(* CODESYS project Flight Simulator_RECOVERED_2024-10-07T14-12-38.project

Project tree, tasks and I/O mapping:
  PLC : HX-CP1S08, Hitachi Industrial Equipment Systems Co., Ltd., order no. HX-CP1S08, version 3.5.8.24
      settings: IP Address = '192.168.137.20'
    application Application
      libraries: Unit Conversion Interfaces, * (Intern); Standard, * (System); VisuDialogs, * (System); CAA Device Diagnosis, 3.5.4.0 (CAA Technical Workgroup); CAA Net Base Services, 3.5.8.10 (CAA Technical Workgroup); NetVarUdp, 3.5.17.0 (System); PRO JSON, 1.0.0.13 (Pro Electric)
      task EtherCAT_Task (cyclic, interval 8 ms, priority 1) calls nothing
      task VISU_TASK (cyclic, interval 200 ms, priority 31) calls VisuElems.Visu_Prg
      task Task (cyclic, interval 20 ms, priority 1) calls main, TcpClient
      global variables gvlSetting
      data type ServoData
      program TcpClient [ST]
      program main [ST]
      visualisation Main
      global variables GVL
    Basic : Basic, Hitachi-IES, version 3.5.8.20
      _16_Digital_Input : 16 Digital Input, Hitachi-IES, version 3.4.0.0
          input  Application.GVL.resetButton : BOOL  // ReserveWord0Type.Bit1
          input  Application.GVL.startButton : BOOL  // ReserveWord0Type.Bit2
          input  Application.GVL.stopButton : BOOL  // ReserveWord0Type.Bit3
          input  Application.GVL.safetySystem : BOOL  // ReserveWord0Type.Bit4
          unmapped channels: ReserveWord0Type, ReserveWord0Type, ReserveWord0Type
      _16_Digital_Output : 16 Digital Output, Hitachi-IES, version 3.4.0.0
          output Application.GVL.LightGreen : BOOL  // ReserveWord0Type.Bit0
          output Application.GVL.LightYellow : BOOL  // ReserveWord0Type.Bit1
          output Application.GVL.LightRed : BOOL  // ReserveWord0Type.Bit2
          unmapped channels: ReserveWord0Type, ReserveWord0Type, ReserveWord0Type
      <Empty>
      <Empty>
      _16_Digital_Input_1 : 16 Digital Input, Hitachi-IES, version 3.4.0.0
          unmapped channels: ReserveWord0Type, ReserveWord0Type, ReserveWord0Type
      <Empty>
      <Empty>
      <Empty>
      <Empty>
      <Empty>
      _16_Digital_Output_1 : 16 Digital Output, Hitachi-IES, version 3.4.0.0
          unmapped channels: ReserveWord0Type, ReserveWord0Type, ReserveWord0Type
    EtherCAT_Master : EtherCAT Master, Festo, version 3.5.16.43
        settings: MasterUseLRW = False; SlaveAutoRestart = True; NetworkName = 'eth2'; NetworkName = "eth2"; SelectNetworkByName = False; EnableTaskMessage = False; SrcAddress1 = 42135; SrcAddress2 = 3137775364; EnableSecondAdapter = False; SrcAddress = [16#A4,16#97,16#BB,16#06,16#A7,16#04]; NetworkName = 'eth2'; NetworkName = "eth2"; SelectNetworkByName = False
      servo_drive_4 : CMMT-AS (point to point), Festo, order no. 5340819, 534082x, 813335x, version 3.5.16.41
          settings: EnableExpertSettings = True; Watchdog register 0400 = 2498; Watchdog register 0410 = 3000; Watchdog register 0420 = 1000; Physical Address of the Slave = 1002; AutoIncr Address of the Slave = 4294967295; FMMU.Global Start Address = 16#02000018; FMMU.Physical Start Address = 16#1000; FMMU.Access = 16#02; FMMU.Global Start Address = 16#01000012; FMMU.Physical Start Address = 16#1100; FMMU.Access = 16#01; FMMU.Global Start Address = 16#00080000; FMMU.StartBit = 1; FMMU.EndBit = 1; FMMU.Physical Start Address = 16#080D; FMMU.Access = 16#01; DC sync0 cycletime = 8000; DC enable = 1; DC sync0 enable = 1; DC sync0 shift time = 0; DC sync1 cycletime = 8000; DC sync1 enable = 0; DC sync1 factor = 'x 1'; DC sync1 shift time = 0
          unmapped channels: Controlword, Modes of operation, Target position, Profile velocity, Target velocity, Target torque, Velocity offset, Torque offset, ---, Statusword, Modes of operation display, Position actual value, Velocity actual value, Torque actual value, Multiturns actual value, ---
      servo_drive_3 : CMMT-AS (point to point), Festo, order no. 5340819, 534082x, 813335x, version 3.5.16.41
          settings: EnableExpertSettings = True; Watchdog register 0400 = 2498; Watchdog register 0410 = 3000; Watchdog register 0420 = 1000; Physical Address of the Slave = 1002; AutoIncr Address of the Slave = 4294967295; FMMU.Global Start Address = 16#02000018; FMMU.Physical Start Address = 16#1000; FMMU.Access = 16#02; FMMU.Global Start Address = 16#01000012; FMMU.Physical Start Address = 16#1100; FMMU.Access = 16#01; FMMU.Global Start Address = 16#00080000; FMMU.StartBit = 1; FMMU.EndBit = 1; FMMU.Physical Start Address = 16#080D; FMMU.Access = 16#01; DC sync0 cycletime = 8000; DC enable = 1; DC sync0 enable = 1; DC sync0 shift time = 0; DC sync1 cycletime = 8000; DC sync1 enable = 0; DC sync1 factor = 'x 1'; DC sync1 shift time = 0
          unmapped channels: Controlword, Modes of operation, Target position, Profile velocity, Target velocity, Target torque, Velocity offset, Torque offset, ---, Statusword, Modes of operation display, Position actual value, Velocity actual value, Torque actual value, Multiturns actual value, ---
      servo_drive_2 : CMMT-AS (point to point), Festo, order no. 5340819, 534082x, 813335x, version 3.5.16.41
          settings: EnableExpertSettings = True; Watchdog register 0400 = 2498; Watchdog register 0410 = 3000; Watchdog register 0420 = 1000; Physical Address of the Slave = 1002; AutoIncr Address of the Slave = 4294967295; FMMU.Global Start Address = 16#02000018; FMMU.Physical Start Address = 16#1000; FMMU.Access = 16#02; FMMU.Global Start Address = 16#01000012; FMMU.Physical Start Address = 16#1100; FMMU.Access = 16#01; FMMU.Global Start Address = 16#00080000; FMMU.StartBit = 1; FMMU.EndBit = 1; FMMU.Physical Start Address = 16#080D; FMMU.Access = 16#01; DC sync0 cycletime = 8000; DC enable = 1; DC sync0 enable = 1; DC sync0 shift time = 0; DC sync1 cycletime = 8000; DC sync1 enable = 0; DC sync1 factor = 'x 1'; DC sync1 shift time = 0
          unmapped channels: Controlword, Modes of operation, Target position, Profile velocity, Target velocity, Target torque, Velocity offset, Torque offset, ---, Statusword, Modes of operation display, Position actual value, Velocity actual value, Torque actual value, Multiturns actual value, ---
      servo_drive_1 : CMMT-AS (point to point), Festo, order no. 5340819, 534082x, 813335x, version 3.5.16.41
          settings: EnableExpertSettings = True; Watchdog register 0400 = 2498; Watchdog register 0410 = 3000; Watchdog register 0420 = 1000; Physical Address of the Slave = 1001; FMMU.Global Start Address = 16#02000000; FMMU.Physical Start Address = 16#1000; FMMU.Access = 16#02; FMMU.Global Start Address = 16#01000000; FMMU.Physical Start Address = 16#1100; FMMU.Access = 16#01; FMMU.Global Start Address = 16#00080000; FMMU.Physical Start Address = 16#080D; FMMU.Access = 16#01; DC sync0 cycletime = 8000; DC enable = 1; DC sync0 enable = 1; DC sync0 shift time = 0; DC sync1 cycletime = 8000; DC sync1 enable = 0; DC sync1 factor = 'x 1'; DC sync1 shift time = 0
          unmapped channels: Controlword, Modes of operation, Target position, Profile velocity, Target velocity, Target torque, Velocity offset, Torque offset, ---, Statusword, Modes of operation display, Position actual value, Velocity actual value, Torque actual value, Multiturns actual value, ---
      servo_drive_6 : CMMT-AS (point to point), Festo, order no. 5340819, 534082x, 813335x, version 3.5.16.41
          settings: EnableExpertSettings = True; Watchdog register 0400 = 2498; Watchdog register 0410 = 3000; Watchdog register 0420 = 1000; Physical Address of the Slave = 1002; AutoIncr Address of the Slave = 4294967295; FMMU.Global Start Address = 16#02000018; FMMU.Physical Start Address = 16#1000; FMMU.Access = 16#02; FMMU.Global Start Address = 16#01000012; FMMU.Physical Start Address = 16#1100; FMMU.Access = 16#01; FMMU.Global Start Address = 16#00080000; FMMU.StartBit = 1; FMMU.EndBit = 1; FMMU.Physical Start Address = 16#080D; FMMU.Access = 16#01; DC sync0 cycletime = 8000; DC enable = 1; DC sync0 enable = 1; DC sync0 shift time = 0; DC sync1 cycletime = 8000; DC sync1 enable = 0; DC sync1 factor = 'x 1'; DC sync1 shift time = 0
          unmapped channels: Controlword, Modes of operation, Target position, Profile velocity, Target velocity, Target torque, Velocity offset, Torque offset, ---, Statusword, Modes of operation display, Position actual value, Velocity actual value, Torque actual value, Multiturns actual value, ---
      servo_drive_5 : CMMT-AS (point to point), Festo, order no. 5340819, 534082x, 813335x, version 3.5.16.41
          settings: EnableExpertSettings = True; Watchdog register 0400 = 2498; Watchdog register 0410 = 3000; Watchdog register 0420 = 1000; Physical Address of the Slave = 1002; AutoIncr Address of the Slave = 4294967295; FMMU.Global Start Address = 16#02000018; FMMU.Physical Start Address = 16#1000; FMMU.Access = 16#02; FMMU.Global Start Address = 16#01000012; FMMU.Physical Start Address = 16#1100; FMMU.Access = 16#01; FMMU.Global Start Address = 16#00080000; FMMU.StartBit = 1; FMMU.EndBit = 1; FMMU.Physical Start Address = 16#080D; FMMU.Access = 16#01; DC sync0 cycletime = 8000; DC enable = 1; DC sync0 enable = 1; DC sync0 shift time = 0; DC sync1 cycletime = 8000; DC sync1 enable = 0; DC sync1 factor = 'x 1'; DC sync1 shift time = 0
          unmapped channels: Controlword, Modes of operation, Target position, Profile velocity, Target velocity, Target torque, Velocity offset, Torque offset, ---, Statusword, Modes of operation display, Position actual value, Velocity actual value, Torque actual value, Multiturns actual value, ---
  libraries: VisuSymbols, 4.1.0.0 (System)
  function block Axis [ST]: enabled, init, doAbort, isReady, doMovement, doReset, getPosition, inError, cycle, isInitialised
  function block signal [ST]: init, cycle
  text list GlobalTextList
  function block Light [ST]: blink, init, cycle, enable
  function block FlightSimulator [ST]: safetyStop, doReset, isEnabled, getPositions, cycle, goNeutralPosition, isReady, doMovement, isInitialised, init, inError, goHomePosition
  data type stateFlightSimulator
*)

// PLC/Application/ServoData
TYPE ServoData :
STRUCT
	positions: ARRAY[1..6] OF JSONVAR;
	speeds: ARRAY[1..6] OF JSONVAR;
END_STRUCT
END_TYPE

// stateFlightSimulator
{attribute 'qualified_only'}
{attribute 'strict'}
TYPE stateFlightSimulator :
(
	error  := 0,
	resetting,
	stopped,
	starting,
	started,
	stopping
);
END_TYPE

// PLC/Application/gvlSetting
{attribute 'qualified_only'}
VAR_GLOBAL CONSTANT
    // Port to use to send data.
	gc_uiPort        : UINT := 32760;
    // IP Address of the computer that hosts the software.
	gc_stIpAddr      : NBS.IP_ADDR := (sAddr := '192.168.137.123');
	// Length of the telegram.
    gc_wMaxTelegram  : INT := 250;
END_VAR

// PLC/Application/GVL
{attribute 'qualified_only'}
VAR_GLOBAL
	// Red light on electrical housing.
	lightRed: BOOL;
	// Yellow light on electrical housing.
	lightYellow: BOOL;
	// Green light on electrical housing.
	lightGreen: BOOL;
	// Reset button on electrical housing.
	resetButton: BOOL := FALSE;
	// Start button on electrical housing.
	startButton: BOOL := FALSE;
	// Stop button on electrical housing.
	stopButton: BOOL := FALSE;
	// Safety system, connected to safety relay.
	safetySystem: BOOL := FALSE;
	// Virtual reset button on HMI.
	resetHMI: BOOL;
	// Virtual start button on HMI.
	startHMI: BOOL;
	// Virtual stop button on HMI.
	stopHMI: BOOL;
	// Virtual toggle button to toggle between tCP data and manual data on HMI.
	useTCPData: BOOL := TRUE;
	// Manual slider velocity input on HMI.
	nextVelocityInput: REAL := 400;
	// Manual slider position input on HMI.
	nextPositionInput: REAL := 0;
	// Flight simulator object.
	FlightSimulator: FlightSimulator;
	// Velocity input from TCP data or HMI data.
	servoVelocities: ARRAY[1..6] OF REAL;
	// Position input from TCP data or HMI data.
	servoPositions: ARRAY[1..6] OF REAL;
	// Current Positions in array format.
	servoPositionsCurrent: ARRAY[1..6] OF REAL;
	// Current Positions in JSON format, used to send back to TCP client.
	currentPositions: ARRAY[1..6] OF JSONVAR;
END_VAR

// PLC/Application/main
PROGRAM main
VAR
	bInit: BOOL := TRUE;
	iCounter : INT;
	bEnabled: BOOL;
	iDataUpdated: INT := 0;
	tonTimer: TON;
END_VAR

IF bInit THEN
	GVL.FlightSimulator.init(
		axis1 := servo_drive_1,
		axis2 := servo_drive_2,
		axis3 := servo_drive_3,
		axis4 := servo_drive_4,
		axis5 := servo_drive_5,
		axis6 := servo_drive_6,
		GVL.lightRed,
		GVL.lightYellow,
		GVL.lightGreen,
		enabled := bEnabled,
		safetySystem := GVL.safetySystem,
		newPositions := GVL.servoPositions,
		newVelocities := GVL.servoVelocities
	);
	bInit := FALSE;
END_IF

// Handle reset buttons.
IF GVL.resetButton OR GVL.resetHMI THEN // blauwe knop
	bEnabled := FALSE;
	GVL.FlightSimulator.doReset();
END_IF

// Handle start buttons.
IF GVL.startButton OR GVL.startHMI THEN // witte knop
	bEnabled := TRUE;
END_IF

// Handle stop buttons
IF GVL.stopButton OR GVL.stopHMI THEN // zwarte knop
	bEnabled := FALSE;
END_IF

// Go through all positions and velocities.
FOR iCounter := 1 TO 6 BY 1 DO 
	IF GVL.useTCPData THEN
		// If TCP data is to be used take data from tcpClient. TCP data can only be toggled via HMI.
		IF tcpClient.parseJSON.Done THEN
			GVL.servoPositions[iCounter] := tcpClient.servoData.positions[iCounter].Number;
			GVL.servoVelocities[iCounter] := tcpClient.servoData.speeds[iCounter].Number;
		END_IF
	ELSE
		// Else take the data from the sliders from the HMI.
		GVL.servoPositions[iCounter] := GVL.nextPositionInput;
		GVL.servoVelocities[iCounter] := GVL.nextVelocityInput;
	END_IF
END_FOR

// Cycle sub functions.
GVL.FlightSimulator.cycle();

// Get current positions, used for TcpClient.
FOR iCounter := 1 TO 6 BY 1 DO
	GVL.currentPositions[iCounter].Number := GVL.FlightSimulator.axis[iCounter].getPosition();
	GVL.servoPositionsCurrent[iCounter] := GVL.FlightSimulator.axis[iCounter].getPosition();
END_FOR

END_PROGRAM

// FlightSimulator
FUNCTION_BLOCK FlightSimulator
VAR_OUTPUT
	// Axis objects.
	axis: ARRAY[1..6] OF Axis;
	// Signal objects.
	signal: signal;
END_VAR
VAR
	// Current state of flight simulator.
	state: stateFlightSimulator;
	// Used in some states to add extra delay.
	bToggle: BOOL;
	// REF to if system should be enabled.
	enabled: REFERENCE TO BOOL;
	// REF to safety system.
	safetySystem: REFERENCE TO BOOL;
	// REF to new positions.
	newPositions: REFERENCE TO ARRAY[1..6] OF REAL;
	// REF to new velocities.
	newVelocities: REFERENCE TO ARRAY[1..6] OF REAL;
END_VAR

METHOD safetyStop : BOOL
VAR
	// Counter to cycle through axis.
	iCounter: UINT;
END_VAR
// Disable all axis.
FOR iCounter := 1 TO 6 BY 1 DO
	THIS^.axis[iCounter].enabled := FALSE;
END_FOR
THIS^.enabled := FALSE;
END_METHOD

METHOD doReset : BOOL
VAR_INPUT
END_VAR
VAR
	// Counter to cycle through axis.
	iCounter: UINT;
END_VAR
THIS^.state := stateFlightSimulator.resetting;
END_METHOD

METHOD isEnabled : BOOL;
VAR_INPUT
END_VAR
VAR
	// Counter to cycle through axis.
	iCounter: INT;
END_VAR
// Check enabled status of all axis, when one is not enabled return with FALSE.
FOR iCounter := 1 TO 6 BY 1 DO
	IF NOT THIS^.axis[iCounter].enabled THEN
		isEnabled := FALSE;
		RETURN;
	END_IF;
END_FOR;

isEnabled := TRUE;
END_METHOD

METHOD getPositions : ARRAY[1..6] OF REAL
VAR_INPUT
END_VAR
VAR
	// Counter to cycle through axis.
	iCounter: INT;
END_VAR
// Write current axis positions
FOR iCounter := 1 TO 6 BY 1 DO
	getPositions[iCounter] := THIS^.axis[iCounter].getPosition();
END_FOR
END_METHOD

METHOD cycle : BOOL
VAR
	// Counter to cycle through axis.
	iCounter: UINT;
END_VAR
// If safety system has been triggered/broken go to error.
IF NOT THIS^.safetySystem THEN
	THIS^.state := stateFlightSimulator.error;
	THIS^.safetyStop();
END_IF

// If any Axis is in error stop all axis.
IF THIS^.inError() AND NOT (THIS^.state = stateFlightSimulator.error) THEN
	IF NOT (THIS^.state = stateFlightSimulator.resetting) THEN
		THIS^.state := stateFlightSimulator.error;
		THIS^.safetyStop();
	END_IF
END_IF

// Reset signal variables.
THIS^.signal.red.enable := FALSE;
THIS^.signal.yellow.enable := FALSE;
THIS^.signal.green.enable := FALSE;
THIS^.signal.red.blink := FALSE;
THIS^.signal.yellow.blink := FALSE;
THIS^.signal.green.blink := FALSE;

// Status case switch.
CASE THIS^.state OF
	stateFlightSimulator.stopped:
		// In STOPPED state:
		// Signal needs to be continuously yellow.
		// Drives needs to be disabled.
		// When enabled go to STARTING state.
		
		// Set signal.
		THIS^.signal.yellow.enable := TRUE;
		
		// Disable drives.
		IF THIS^.isEnabled() THEN
			FOR iCounter := 1 TO 6 BY 1 DO
				Axis[iCounter].enabled := FALSE;
			END_FOR
		END_IF
		
		// If flightsim is enabled go to STARTING state.
		IF THIS^.enabled THEN
			THIS^.state := stateFlightSimulator.starting;
		END_IF
		
	stateFlightSimulator.starting:
		// In STARTING state:
		// Signal needs to be blinking green.
		// Drives needs to be enabled.
		// Once enabled go to neutral position.
		// Once in neutral position go to STARTED state.
	
		// Set signal.
		THIS^.signal.green.enable := TRUE;
		THIS^.signal.green.blink := TRUE;
		
		// Start Axises.
		IF NOT THIS^.isEnabled() THEN
			FOR iCounter := 1 TO 6 BY 1 DO
				Axis[iCounter].enabled := TRUE;
			END_FOR
		END_IF
		
		IF THIS^.isEnabled() AND THIS^.isReady() THEN
			IF NOT bToggle THEN
				// Move pistons to neutral position.
				THIS^.goNeutralPosition();
				bToggle := TRUE;
			ELSE
				// When position has been reached go to started state.
				bToggle := FALSE;
				THIS^.state := stateFlightSimulator.started;
			END_IF	
		END_IF
		
	stateFlightSimulator.started:
		// In STARTED state:
		// Signal needs to be continuously green.
		// When at least one of the drives goes to disabled go to ERROR state.
		// Do movement.
		// When not enabled go to STOPPING state.
	
		// Set signal.
		THIS^.signal.green.enable := TRUE;
		
		// If drives are disabled somehow go to error.
		IF NOT THIS^.isEnabled() THEN
			THIS^.state := stateFlightSimulator.error;
		END_IF
		
		// Do movement.
		THIS^.doMovement(THIS^.newPositions, THIS^.newVelocities);
		
		// If flightsim is disabled go to STOPPING state.
		IF NOT THIS^.enabled THEN
			THIS^.state := stateFlightSimulator.stopping;
		END_IF
		
	stateFlightSimulator.stopping:
		// In STOPPING state:
		// Signal needs to be blinking green.
		// Drives needs to be enabled.
		// Once enabled go to home position.
		// Once in home position go to STOPPED state.
	
		// Set signal.
		THIS^.signal.green.enable := TRUE;
		THIS^.signal.green.blink := TRUE;
		
		// Enable drives if not enabled yet.
		IF NOT THIS^.isEnabled() THEN
			FOR iCounter := 1 TO 6 BY 1 DO
				Axis[iCounter].enabled := TRUE;
			END_FOR
		END_IF
		
		IF THIS^.isEnabled() THEN
			IF NOT bToggle THEN
				// Move pistons to home position.
				THIS^.goHomePosition();
				bToggle := TRUE;
			ELSE
				IF THIS^.isReady() THEN
					// When position has been reached go to stopped state.
					bToggle := FALSE;
					THIS^.state := stateFlightSimulator.stopped;
				END_IF
			END_IF
		END_IF
		
	stateFlightSimulator.error:
		// In ERROR state:
		// Signal needs to be blinking red.
		
		// Set signal.
		THIS^.signal.red.enable := TRUE;
		THIS^.signal.red.blink := TRUE;
		
	stateFlightSimulator.resetting:
		// In RESETTING state:
		// Signal needs to be blinking yellow.
		// If in error drives needs to be reset.
		// Else go to home and go to STOPPED state.
	
		// Set signal.
		THIS^.signal.yellow.enable := TRUE;
		THIS^.signal.yellow.blink := TRUE;
		
		IF THIS^.inError() THEN
			// Reset drives.
			FOR iCounter := 1 TO 6 BY 1 DO
				Axis[iCounter].doReset();
			END_FOR
		ELSE
			// Enable drives if not enabled yet.
			IF NOT THIS^.isEnabled() THEN
				FOR iCounter := 1 TO 6 BY 1 DO
					Axis[iCounter].enabled := TRUE;
				END_FOR
			END_IF
			
			IF THIS^.isEnabled() THEN
				IF NOT bToggle THEN
					// Move pistons to home position.
					THIS^.goHomePosition();
					bToggle := TRUE;
				ELSE
					IF THIS^.isReady() THEN
						// When position has been reached go to stopped state.
						bToggle := FALSE;
						THIS^.state := stateFlightSimulator.stopped;
					END_IF
				END_IF
			END_IF
		END_IF
END_CASE

// Cycle Axis classes.
FOR iCounter := 1 TO 6 BY 1 DO
	THIS^.axis[iCounter].cycle();
END_FOR
// Cycle signal class.
THIS^.signal.cycle();
END_METHOD

METHOD goNeutralPosition : BOOL
VAR
	// Counter to cycle through axis.
	iCounter: INT;
END_VAR
IF THIS^.isReady() THEN
	FOR iCounter := 1 TO 6 BY 1 DO
		THIS^.axis[iCounter].doMovement(position := 200, velocity := 25, continuousUpdate:=FALSE);
	END_FOR
END_IF
END_METHOD

METHOD isReady : BOOL
VAR_INPUT
END_VAR
VAR
	// Counter to cycle through axis.
	iCounter: INT;
END_VAR
// Check ready status of all axis, when one is not ready return with FALSE.
FOR iCounter := 1 TO 6 BY 1 DO
	IF NOT THIS^.axis[iCounter].isReady() THEN
		isReady := FALSE;
		RETURN;
	END_IF;
END_FOR;

isReady := TRUE;
END_METHOD

METHOD doMovement : BOOL
VAR_INPUT
	positions : ARRAY[1..6] OF REAL;
	speeds : ARRAY[1..6] OF REAL;
END_VAR
VAR
	// Counter to cycle through axis.
	iCounter: INT;
	// Var that says its safe to execute this command, will be lowered in the FOR loop check.
	bSafe: BOOL := TRUE;
END_VAR
FOR iCounter := 1 TO 6 BY 1 DO
	// If any of the positions are larger than 390 or smaller than 10 don't execute the command.
	IF positions[iCounter] > 390 OR positions[iCounter] < 10 THEN
		bSafe := FALSE;
	END_IF
	
	// If any of the velocities are larger than 401 or smaller than 0 don't execute the command.
	IF speeds[iCounter] >= 401 OR speeds[iCounter] < 0 THEN
		bSafe := FALSE;
	END_IF
END_FOR

IF bSafe THEN
	FOR iCounter := 1 TO 6 BY 1 DO
		Axis[iCounter].doMovement(position:=positions[iCounter], velocity:=speeds[iCounter], continuousUpdate:=TRUE);
	END_FOR
END_IF
END_METHOD

METHOD isInitialised : BOOL
VAR_INPUT
END_VAR
VAR
	// Counter to cycle through axis.
	iCounter: INT;
END_VAR
// Check if all axis are initialised, when one is not initialised return with FALSE.
FOR iCounter := 1 TO 6 BY 1 DO
	IF NOT THIS^.axis[iCounter].isInitialised() THEN
		isInitialised := FALSE;
		RETURN;
	END_IF;
END_FOR;

isInitialised := TRUE;
END_METHOD

METHOD init : BOOL
VAR_INPUT
	axis1: REFERENCE TO AXIS_REF_FESTO;
	axis2: REFERENCE TO AXIS_REF_FESTO;
	axis3: REFERENCE TO AXIS_REF_FESTO;
	axis4: REFERENCE TO AXIS_REF_FESTO;
	axis5: REFERENCE TO AXIS_REF_FESTO;
	axis6: REFERENCE TO AXIS_REF_FESTO;
	lightRed: REFERENCE TO BOOL;
	lightYellow: REFERENCE TO BOOL;
	lightGreen: REFERENCE TO BOOL;
	enabled: REFERENCE TO BOOL;
	// When this variable is HIGH it means that the safety system is active.
	// This means none of it's safety systems has been triggered.
	safetySystem: REFERENCE TO BOOL;
	newPositions: REFERENCE TO ARRAY[1..6] OF REAL;
	newVelocities: REFERENCE TO ARRAY[1..6] OF REAL;
END_VAR
THIS^.axis[1].init(axis1);
THIS^.axis[2].init(axis2);
THIS^.axis[3].init(axis3);
THIS^.axis[4].init(axis4);
THIS^.axis[5].init(axis5);
THIS^.axis[6].init(axis6);

THIS^.signal.init(lightRed, lightYellow, lightGreen);

THIS^.enabled REF= enabled;
THIS^.safetySystem REF= safetySystem;

THIS^.newPositions REF= newPositions;
THIS^.newVelocities REF= newVelocities;
END_METHOD

METHOD inError : BOOL
VAR
	// Counter to cycle through axis.
	iCounter: INT;
END_VAR
// Check error status of all axis, when one is in error return with TRUE.
FOR iCounter := 1 TO 6 BY 1 DO
	IF THIS^.axis[iCounter].inError() THEN
		inError := TRUE;
		RETURN;
	END_IF;
END_FOR;

InError := FALSE;
END_METHOD

METHOD goHomePosition : BOOL
VAR
	// Counter to cycle through axis.
	iCounter: INT;
END_VAR
// Abort current movement action.
FOR iCounter := 1 TO 6 BY 1 DO
	THIS^.axis[iCounter].doAbort();
END_FOR

IF THIS^.isReady() THEN
	FOR iCounter := 1 TO 6 BY 1 DO
		THIS^.axis[iCounter].doMovement(position := 10, velocity := 25, continuousUpdate:=FALSE);
	END_FOR
END_IF
END_METHOD

END_FUNCTION_BLOCK

// Axis
FUNCTION_BLOCK Axis
VAR
	// Power stage of the servo drive.
	MC_Power: MC_Power_Festo;
	// Reset object to reset servo drive.
	MC_Reset: MC_Reset_Festo;
	// Move absolute object to move the servo.
	MC_MoveAbsolute: MC_MoveAbsolute_Festo;
	// Read object to read current position.
	MC_ReadActualPosition: MC_ReadActualPosition_Festo;
	// Read status object to read current status of servo drive.
	MC_ReadStatus: MC_ReadStatus_Festo;
	
	// REF to axis.
	axis: REFERENCE TO AXIS_REF_FESTO;
	// Allow move orders to be overwritten by new moveorders.
	continuousUpdate: BOOL := FALSE;
	// Execute a move order.
	execute: BOOL := FALSE;
	// Drive is enabled.
	isEnabled: BOOL := FALSE;
	// Drive is in error.
	error: BOOL := FALSE;
	// Drive is beign reset, toggle bit.
	reset: BOOL := FALSE;
	// Requested position of servo.
	position: REAL := 0;
	// Requested velocity of servo.
	velocity: REAL := 0;
	// Acceleration of servo.
	acceleration: REAL := 5000;
	// Deceleration of servo.
	deceleration: REAL := 5000;
	// Jerk of servo.
	jerk: REAL := 15000;
END_VAR

PROPERTY enabled : BOOL
GET
enabled := THIS^.isEnabled AND (NOT THIS^.MC_ReadStatus.Disabled);
END_GET
SET
THIS^.isEnabled := enabled;
END_SET
END_PROPERTY

METHOD init : BOOL
VAR_INPUT
	axis : REFERENCE TO AXIS_REF_FESTO;
END_VAR
// This function references the servo drive to the instance of the function block.
THIS^.axis REF= axis;
END_METHOD

METHOD doAbort : BOOL
VAR_INPUT
END_VAR
THIS^.execute := FALSE;
END_METHOD

METHOD isReady : BOOL
VAR_INPUT
END_VAR
// Axis is ready when in standstill and not been given an execution order.
isReady := THIS^.MC_ReadStatus.Standstill AND NOT THIS^.execute;
END_METHOD

METHOD doMovement : BOOL
VAR_INPUT
	velocity: REAL := 0;
	position: REAL := 0;
	continuousUpdate: BOOL := FALSE;
END_VAR
// Only do movements when drive is started.
IF THIS^.isEnabled THEN
	THIS^.position := position;
	THIS^.velocity := velocity; 
	THIS^.continuousUpdate := continuousUpdate;
	THIS^.execute := TRUE;
	DoMovement := TRUE;		// return
ELSE
	THIS^.execute := FALSE;
	DoMovement := FALSE;	// return
END_IF;
END_METHOD

METHOD doReset
THIS^.reset := TRUE;
END_METHOD

METHOD getPosition : REAL
VAR_INPUT
END_VAR
IF THIS^.MC_ReadActualPosition.Valid OR (NOT THIS^.MC_ReadActualPosition.Error) THEN
	getPosition := THIS^.MC_ReadActualPosition.Position;
ELSE
	getPosition := -1;
END_IF
END_METHOD

METHOD inError : BOOL
VAR_INPUT
END_VAR
inError := THIS^.error;
END_METHOD

METHOD cycle : BOOL
VAR_INPUT
END_VAR
// Read drive status first
MC_ReadStatus(
	axis := THIS^.axis, 
	Enable := TRUE
);

// Set drive to error if an error occurs.
IF THIS^.MC_ReadStatus.ErrorStop OR THIS^.MC_ReadStatus.Error THEN
	THIS^.error := TRUE;
END_IF

// Function block to enable the drive.
THIS^.MC_Power(
	axis := THIS^.axis,
	Enable := THIS^.isEnabled
);

// Function block to reset the drive.
THIS^.MC_Reset(
	axis := THIS^.axis,
	Execute := THIS^.reset
);

// Reset the reset variable
IF (THIS^.MC_Reset.Done AND THIS^.reset) OR THIS^.MC_Reset.Error THEN
	THIS^.reset := FALSE;
	THIS^.error := FALSE;
END_IF

// Reset execute when movement is done.
IF (THIS^.MC_MoveAbsolute.Done AND NOT THIS^.continuousUpdate) OR THIS^.MC_MoveAbsolute.CommandAborted OR THIS^.error THEN
	THIS^.execute := FALSE;
END_IF

// Reset the move function if it's in error.
IF NOT THIS^.MC_MoveAbsolute.Error THEN
	// Function block to move the drive.
	THIS^.MC_MoveAbsolute(
		axis := THIS^.axis,
		Execute := THIS^.execute,
		ContinuousUpdate := THIS^.continuousUpdate,
		position := THIS^.position,
		velocity := THIS^.velocity,
		acceleration := THIS^.acceleration,
		deceleration := THIS^.deceleration,
		jerk := THIS^.jerk
	);
ELSE
	THIS^.MC_MoveAbsolute(axis := THIS^.axis, Execute := FALSE);
END_IF;

// Function block to read the drives current position.
THIS^.MC_ReadActualPosition(
	axis := THIS^.axis,
	Enable := TRUE
);
END_METHOD

METHOD isInitialised : BOOL
VAR_INPUT
END_VAR
isInitialised := THIS^.MC_ReadStatus.Valid;
END_METHOD

END_FUNCTION_BLOCK

// signal
FUNCTION_BLOCK signal
VAR_INPUT
	// Red light.
	red: light;
	// Yellow light.
	yellow: light;
	// Green light.
	green: light;
END_VAR
VAR
	
	// TON.
	clockTON: TON;
	// TOF.
	clockTOF: TOF;
	// Current clock state.
	clock: BOOL;
END_VAR

METHOD init : BOOL
VAR_INPUT
	red: REFERENCE TO BOOL;
	yellow: REFERENCE TO BOOL;
	green: REFERENCE TO BOOL;
END_VAR
VAR
END_VAR
THIS^.red.init(red, clock);
THIS^.yellow.init(yellow, clock);
THIS^.green.init(green, clock);
END_METHOD

METHOD cycle : BOOL
VAR_INPUT
END_VAR
clockTON(IN:= NOT clockTOF.Q, PT:=T#500MS);
clockTOF(IN:= clockTON.Q, PT:=T#500MS);
THIS^.clock := clockTOF.Q;

// Cycle light objects.
THIS^.red.cycle();
THIS^.yellow.cycle();
THIS^.green.cycle();
END_METHOD

END_FUNCTION_BLOCK

// Light
FUNCTION_BLOCK Light
VAR
	light: REFERENCE TO BOOL;
	clock: REFERENCE TO BOOL;
	
	enabled: BOOL := FALSE;
	blinking: BOOL := FALSE;
END_VAR

PROPERTY blink : BOOL
SET
THIS^.blinking := blink;
END_SET
GET
blink := THIS^.blinking;
END_GET
END_PROPERTY

METHOD init : BOOL
VAR_INPUT
	light: REFERENCE TO BOOL;
	clock: REFERENCE TO BOOL;
END_VAR
VAR
END_VAR
THIS^.light REF= light;
THIS^.clock REF= clock;
END_METHOD

METHOD cycle : BOOL
VAR_INPUT
END_VAR
IF THIS^.enabled THEN
	IF THIS^.blinking THEN
		// If blinking is enabled, turn light on or off depending on clock state.
		IF THIS^.clock THEN
			THIS^.light := TRUE;
		ELSE
			THIS^.light := FALSE;
		END_IF
	ELSE
			THIS^.light := TRUE;
	END_IF
ELSE
	THIS^.light := FALSE;
END_IF
END_METHOD

PROPERTY enable : BOOL
GET
enable := THIS^.enabled;
END_GET
SET
THIS^.enabled := enable;
END_SET
END_PROPERTY

END_FUNCTION_BLOCK

// PLC/Application/TcpClient
PROGRAM TcpClient
VAR

    // Client object that connects to client machine.
	fbTcpClient   : NBS.TCP_Client;
    // Read object that reads incomming data from client machine.
	fbTcpRead     : NBS.TCP_Read;
    // Write object that writes data to client machine.
	fbTcpWrite    : NBS.TCP_Write;
	
	// TON object for reset delay.
	tonResetDelay: TON;
	// Received telegram from Read object.
	received      : STRING(gvlSetting.gc_wMaxTelegram);
	// Sent telegram to Write object.
	sent          : STRING(gvlSetting.gc_wMaxTelegram);
	// JSON Parser object to parse read data.
	parseJSON     : JSON_TO_STRUCT;
	// JSON Composer object to compose data to write.
	composeJSON   : STRUCT_TO_JSON;
	// Struct that stores the received data in usable arrays.
	servoData     : ServoData;
    // Make connection.
	xConnect      : BOOL := TRUE;
	// Do composing.
	xCompose: BOOL;
	// Do write action.
	xWrite: BOOL;
	// Do parsing
	xParse: BOOL;
 
    // Do read action.
	xRead         : BOOL;
    // Size of read data telegram.
	udiRead       : UDINT;
	// Timeout in µs.
	udiTimeOut: UDINT := 500000;
	
	
	udiVal        : UDINT;
    pudiVal       : POINTER TO BYTE;
    iIndex        : INT;
	xMissingAck   : BOOL;
    udiResult     : UDINT;
    udiLastAck    : UDINT;
    udiNow        : UDINT;
END_VAR

fbTcpClient(xEnable := xConnect, ipAddr := gvlSetting.gc_stIpAddr, uiPort := gvlSetting.gc_uiPort, udiTimeOut := udiTimeOut);

// Run when connection is active.
IF fbTcpClient.xActive AND GVL.FlightSimulator.isInitialised() THEN
	
	IF fbTcpWrite.xDone THEN
		xWrite := FALSE;
	ELSIF NOT fbTcpWrite.xBusy THEN
		IF composeJSON.Done AND composeJSON.Execute THEN
			xCompose := FALSE;
			xWrite := TRUE;
		ELSIF (NOT composeJSON.Busy) THEN
			   xCompose := TRUE;
			   xWrite := FALSE;
		END_IF
	END_IF
	
	composeJSON(
		Execute:= xCompose,
		JSONString:= ADR(sent),
		JSONStringSize:= SIZEOF(sent),
		JSONVars:= ADR(GVL.currentPositions),
		NumberOfVars:= SIZEOF(GVL.currentPositions) / SIZEOF(JSONVAR)
	); 
	fbTcpWrite(xExecute := xWrite, hConnection := fbTcpClient.hConnection, udiTimeOut := udiTimeOut, szSize := SIZEOF(sent), pData := ADR(sent));
	
	IF (NOT fbTcpRead.xBusy) AND (NOT parseJSON.Busy) THEN
		xRead := TRUE;
	ELSIF fbTcpRead.xReady THEN
		xRead := FALSE;
		xParse := TRUE;
	ELSIF (NOT parseJSON.Busy) THEN
		xParse := FALSE;
	END_IF

	parseJSON(
		Execute := xParse,
		JSONString:= ADR(received),
		JSONStringSize:= SIZEOF(received),
		JSONVars:= ADR(servoData),
		NumberOfVars:= SIZEOF(servoData) / SIZEOF(JSONVAR)
	);
	fbTcpRead(xEnable := xRead, hConnection := fbTcpClient.hConnection, szSize := SIZEOF(received), pData := ADR(received), szCount => udiRead);
	
END_IF

// Reset connection when connection has stopped.
IF (NOT xConnect) THEN
	// Reset all variables.
	xConnect := FALSE;
	xWrite := FALSE;
	xCompose := FALSE;
	fbTcpWrite(xExecute := FALSE);
	xRead := FALSE;
	xParse := FALSE;
	fbTcpRead(xEnable := FALSE);
	received := '';
	sent := '';
	// Delay reset for 3 sec.
	tonResetDelay(IN:=TRUE, PT:=T#3S);
	IF (tonResetDelay.Q) THEN
		tonResetDelay(IN:=FALSE);
		xConnect := TRUE;
	END_IF
	
END_IF

IF fbTcpClient.xDone AND xConnect THEN
	xConnect := FALSE;
END_IF

// Stop connection when in error.
IF fbTcpClient.xError OR fbTcpWrite.xError OR fbTcpRead.xError THEN
	xConnect := FALSE;
	fbTcpWrite(xExecute := FALSE);
END_IF

END_PROGRAM

// PLC/Application/Main
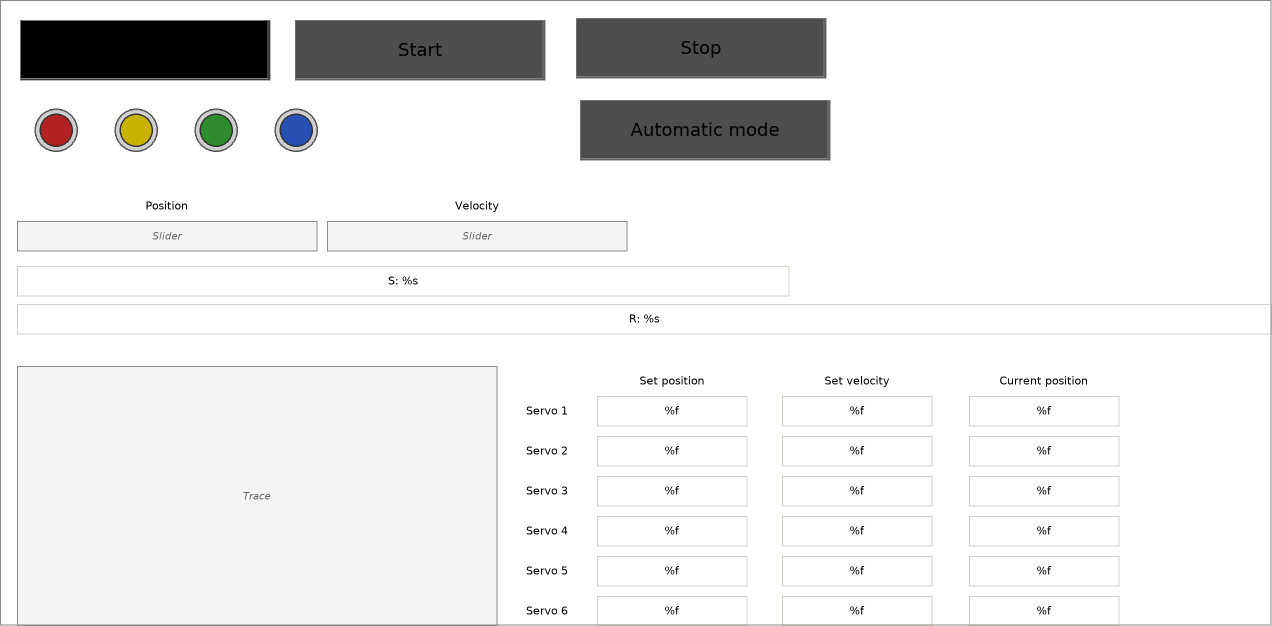
VISUALIZATION Main  // 1272x626
    Button (20,20 250x60), "Reset"
        tap GVL.resetHMI
    Button (295,20 250x60), "Start"
        tap GVL.startHMI
    Slider (17,221 300x30), variable: GVL.nextPositionInput, scale 10..390
    Button (580,100 250x60), "Automatic mode"
        toggle GVL.usetcpdata
    Slider (327,221 300x30), variable: GVL.nextVelocityInput, scale 0..400
    Button (576,18 250x60), "Stop"
        tap GVL.stopHMI
    Lamp1 (191,105 50x50), variable: GVL.lightGreen, style: Lamp-Lamp1-Green
    Lamp1 (31,105 50x50), variable: GVL.lightRed, style: Lamp-Lamp1-Red
    Lamp1 (111,105 50x50), variable: GVL.lightYellow, style: Lamp-Lamp1-Yellow
    Textfield (17,266 772x30), "S: %s", text variable: TcpClient.sent
    Textfield (17,304 1255x30), "R: %s", text variable: TcpClient.received
    Textfield (597,396 150x30), "%f", text variable: GVL.servoPositions[1]
        OnMouseClick: write the text variable via InputWithLimits, min 0, max 400
    Textfield (597,436 150x30), "%f", text variable: GVL.servoPositions[2]
        OnMouseClick: write the text variable via InputWithLimits, min 0, max 400
    Textfield (597,476 150x30), "%f", text variable: GVL.servoPositions[3]
        OnMouseClick: write the text variable via InputWithLimits, min 0, max 400
    Textfield (597,516 150x30), "%f", text variable: GVL.servoPositions[4]
        OnMouseClick: write the text variable via InputWithLimits, min 0, max 400
    Textfield (597,556 150x30), "%f", text variable: GVL.servoPositions[5]
        OnMouseClick: write the text variable via InputWithLimits, min 0, max 400
    Textfield (597,596 150x30), "%f", text variable: GVL.servoPositions[6]
        OnMouseClick: write the text variable via InputWithLimits, min 0, max 400
    Textfield (782,396 150x30), "%f", text variable: GVL.servoVelocities[1]
        OnMouseClick: write the text variable via InputWithLimits, min 0, max 400
    Textfield (782,436 150x30), "%f", text variable: GVL.servoVelocities[2]
        OnMouseClick: write the text variable via InputWithLimits, min 0, max 400
    Textfield (782,476 150x30), "%f", text variable: GVL.servoVelocities[3]
        OnMouseClick: write the text variable via InputWithLimits, min 0, max 400
    Textfield (782,516 150x30), "%f", text variable: GVL.servoVelocities[4]
        OnMouseClick: write the text variable via InputWithLimits, min 0, max 400
    Textfield (782,556 150x30), "%f", text variable: GVL.servoVelocities[5]
        OnMouseClick: write the text variable via InputWithLimits, min 0, max 400
    Textfield (782,596 150x30), "%f", text variable: GVL.servoVelocities[6]
        OnMouseClick: write the text variable via InputWithLimits, min 0, max 400
    Label (597,366 150x30), "Set position"
    Label (782,366 150x30), "Set velocity"
    Label (497,396 100x30), "Servo 1"
    Label (497,436 100x30), "Servo 2"
    Label (497,476 100x30), "Servo 3"
    Label (497,516 100x30), "Servo 4"
    Label (497,556 100x30), "Servo 5"
    Label (497,596 100x30), "Servo 6"
    Lamp1 (271,105 50x50), variable: GVL.FlightSimulator.isReady(), style: Lamp-Lamp1-Blue
    Trace (17,366 480x260)
    Textfield (969,396 150x30), "%f", text variable: GVL.servoPositionsCurrent[1]
        OnMouseClick: write the text variable via InputWithLimits, min 0, max 400
    Textfield (969,436 150x30), "%f", text variable: GVL.servoPositionsCurrent[2]
        OnMouseClick: write the text variable via InputWithLimits, min 0, max 400
    Textfield (969,476 150x30), "%f", text variable: GVL.servoPositionsCurrent[3]
        OnMouseClick: write the text variable via InputWithLimits, min 0, max 400
    Textfield (969,516 150x30), "%f", text variable: GVL.servoPositionsCurrent[4]
        OnMouseClick: write the text variable via InputWithLimits, min 0, max 400
    Textfield (969,556 150x30), "%f", text variable: GVL.servoPositionsCurrent[5]
        OnMouseClick: write the text variable via InputWithLimits, min 0, max 400
    Textfield (969,596 150x30), "%f", text variable: GVL.servoPositionsCurrent[6]
        OnMouseClick: write the text variable via InputWithLimits, min 0, max 400
    Label (969,366 150x30), "Current position"
    Label (92,191 150x30), "Position"
    Label (402,191 150x30), "Velocity"
END_VISUALIZATION
